(* IEC 61131-3 sources: CodesysTest/alpha/export/Pro18_1174_Win10.dev/Plc Logic/Application/Motors/Festo/FB_FestoMotor.pou/Moving.prop, 1 file *)

(* ---- Get.pm.st ---- *)
(*#-#-#-#-#-#-#-#-#-#---Declaration---#-#-#-#-#-#-#-#-#-#-#-#-#*)

VAR
END_VAR
(*#-#-#-#-#-#-#-#-#-#---Implementation---#-#-#-#-#-#-#-#-#-#-#-#-#*)

Moving := CRTL_Axis.DriveIsMoving;
